(* CODESYS project Parcial2_CPI.project

Project tree, tasks and I/O mapping:
  Device : CODESYS Control Win V3 x64, 3S - Smart Software Solutions GmbH, version 3.5.17.10
    application Application
      libraries: Standard, * (System); CmpBitmapPool, * (System); Util, * (System)
      task MainTask (cyclic, interval t#20ms, priority 1) calls PLC_PRG
      task Simu (cyclic, interval t#20ms, priority 1) calls POU, BOTTLE_SIM
      task VISU_TASK (cyclic, interval 100 ms, priority 31) calls VisuElems.Visu_Prg
      global variables GVL
      program PLC_PRG [ST]
      SIMULACION/
        program BOTTLE_SIM [ST]
        image pool ImagePool
        OBJECTS_METHODS/
          data type BOTTLE_structure
          function colision_detection [ST]
          function modulo [ST]
        program POU [ST]
      visualisation Visualization
      Symbols
      function block AUTO_BF [ST]
      function block MANUAL_BF [ST]
    Ethernet : Ethernet, 3S - Smart Software Solutions GmbH, version 3.5.17.0
        settings: IPAddress = [10,70,28,96]; SubnetMask = [255,255,224,0]; GatewayAddress = [10,70,0,1]; MACAddress = [16#F8,16#5E,16#A0,16#06,16#18,16#05]; NetworkInterfaceName = 'Wi-Fi'; NetworkInterfaceName = "Wi-Fi"; SaveCommunicationSettings = FALSE
      ModbusTCP_Slave_Device : ModbusTCP Slave Device, 3S - Smart Software Solutions GmbH, version 3.5.17.0
          input  Application.PLC_PRG.BOTON_STOP : BOOL  // Registros Holding.Registros Holding.Bit0
          input  Application.PLC_PRG.BOTON_MANUAL : BOOL  // Registros Holding.Registros Holding.Bit1
          input  Application.PLC_PRG.BOTON_AUTO : BOOL  // Registros Holding.Registros Holding.Bit2
          input  Application.BAC1_HMI : BOOL  // Registros Holding.Registros Holding.Bit3
          input  Application.BAC2_HMI : BOOL  // Registros Holding.Registros Holding.Bit4
          input  Application.BABanda_HMI : BOOL  // Registros Holding.Registros Holding.Bit5
          input  Application.BAProducto_HMI : BOOL  // Registros Holding.Registros Holding.Bit6
          input  Application.BAMezclador_HMI : BOOL  // Registros Holding.Registros Holding.Bit7
          input  Application.BADosificacion_HMI : BOOL  // Registros Holding.Registros Holding.Bit8
          input  Application.BOTTLE_SIM.agregar : BOOL  // Registros Holding.Registros Holding.Bit9
          input  Application.BOTTLE_SIM.eliminar : BOOL  // Registros Holding.Registros Holding.Bit10
          output Application.PLC_PRG.PARADA : BOOL  // Registros Input.Registros Input.Bit0
          output Application.PLC_PRG.MANUAL : BOOL  // Registros Input.Registros Input.Bit1
          output Application.PLC_PRG.AUTO : BOOL  // Registros Input.Registros Input.Bit2
          output Application.BAC1_HMI : BOOL  // Registros Input.Registros Input.Bit3
          output Application.BAC2_HMI : BOOL  // Registros Input.Registros Input.Bit4
          output Application.BABanda_HMI : BOOL  // Registros Input.Registros Input.Bit5
          output Application.BAProducto_HMI : BOOL  // Registros Input.Registros Input.Bit6
          output Application.BAMezclador_HMI : BOOL  // Registros Input.Registros Input.Bit7
          output Application.BADosificacion_HMI : BOOL  // Registros Input.Registros Input.Bit8
          unmapped channels: Registros Holding, Registros Input
  libraries: VisuSymbols, 3.5.17.0 (System)
  text list GlobalTextList
  5ce3da45-db07-42e7-a21c-a00fff4ed8f6|imagenes\P1.png
  5ce3da45-db07-42e7-a21c-a00fff4ed8f6|imagenes\P2.png
  5ce3da45-db07-42e7-a21c-a00fff4ed8f6|imagenes\P3.png
  5ce3da45-db07-42e7-a21c-a00fff4ed8f6|imagenes\P4.png
  5ce3da45-db07-42e7-a21c-a00fff4ed8f6|imagenes\P5.png
  5ce3da45-db07-42e7-a21c-a00fff4ed8f6|imagenes\P6.png
  5ce3da45-db07-42e7-a21c-a00fff4ed8f6|imagenes\WaterEmpty.png
  5ce3da45-db07-42e7-a21c-a00fff4ed8f6|imagenes\WaterFilled.png
  5ce3da45-db07-42e7-a21c-a00fff4ed8f6|imagenes\banda.png
  5ce3da45-db07-42e7-a21c-a00fff4ed8f6|imagenes\Cilindro.png
  5ce3da45-db07-42e7-a21c-a00fff4ed8f6|imagenes\Fence.png
  5ce3da45-db07-42e7-a21c-a00fff4ed8f6|imagenes\fondo.png
  5ce3da45-db07-42e7-a21c-a00fff4ed8f6|imagenes\prod2.png
  5ce3da45-db07-42e7-a21c-a00fff4ed8f6|imagenes\prod3.png
  5ce3da45-db07-42e7-a21c-a00fff4ed8f6|imagenes\prod1.png
*)

// Device/Application/SIMULACION/OBJECTS_METHODS/BOTTLE_structure
TYPE BOTTLE_structure :
STRUCT
	empty : BOOL := TRUE; // solid image box
	filled : BOOL := TRUE; // glued image box
	
	pos_x: INT := 0; // x position
	posr_x: REAL := 0; // x position
	
	mvx: REAL := 0.3; // velocidad de movimiento en x
	vx: REAL; // velocidad en x
	
	t_llenado: TON;
END_STRUCT
END_TYPE

// Device/Application/GVL
VAR_GLOBAL
	//MOTORES TRIFASICOS
	BAProducto: BOOL := FALSE; // Señal para encender el motoreductor trifasico elevador del producto
	BAMezclador: BOOL := FALSE; // Señal para encender el motoreductor trifasico de mezclado en la tolva
	BADosificacion: BOOL := FALSE; // Señal para encender el motoreductor trifasico de giro del tornillo de dosificación
	BABanda: BOOL := FALSE; // Señal para encender el motoreductor trifasico de la banda transportadora
	
	//CILINDRO 1 (QUE DETIENE LOS RECIPIENTES QUE VAN A ENTRAR AL PUNTO DE DOSIFICACIÓN)
	BAC1 : BOOL := FALSE; // Señal de avance para el cilindro 1
	SFC1 : BOOL; // Señal de posición final para el cilindro 1
	SIC1 : BOOL; // Señal de posición inicial para el cilindro 1
	
	//CILINDRO 2 (QUE DETIENE EL RECIPIENTE EN EL PUNTO DE DOSIFICACIÓN)
	BAC2 : BOOL := FALSE; // Señal de avance para el cilindro 2
	SFC2 : BOOL; // Señal de posición final para el cilindro 2
	SIC2 : BOOL; // Señal de posición inicial para el cilindro 2
	
	//SENSOR DE PRESENCIA
	SL: BOOL := FALSE; //Sensor de botella en la zona de llenado
	
	//SENSOR DE NIVEL
	NT: INT; //Sensor de 10 bits del nivel de la tolva 
	NTD: BOOL; //Sensor digital del nivel de la tolva (activo cuando el nivel es mayor a 95%)
	
	//HMI
	BAC1_HMI: BOOL;
	BAC2_HMI: BOOL;
	BAProducto_HMI: BOOL;
	BAMezclador_HMI: BOOL;
	BADosificacion_HMI: BOOL;
	BABanda_HMI: BOOL;
	
END_VAR

// Device/Application/PLC_PRG
PROGRAM PLC_PRG
VAR

	PARADA: BOOL := TRUE;
	MANUAL: BOOL;
	AUTO: BOOL;
	BOTON_STOP: BOOL;
	BOTON_MANUAL: BOOL;
	BOTON_AUTO: BOOL;
	
	AUTO1 : AUTO_BF;
	MANUAL1 : MANUAL_BF;
	
END_VAR


IF PARADA AND BOTON_MANUAL THEN
	PARADA := FALSE;
	AUTO := FALSE;
	MANUAL:= TRUE;
	
ELSIF MANUAL AND BOTON_AUTO THEN
	PARADA := FALSE;
	MANUAL:= FALSE;
	AUTO := TRUE;

ELSIF MANUAL AND BOTON_STOP THEN
	PARADA := TRUE;
	AUTO := FALSE;
	MANUAL:= FALSE;

ELSIF AUTO AND BOTON_STOP THEN
	PARADA := TRUE;
	AUTO := FALSE;
	MANUAL:= FALSE;
	
ELSIF PARADA AND BOTON_AUTO THEN
	PARADA := FALSE;
	AUTO := TRUE;
	MANUAL:= FALSE;
	
END_IF

IF PARADA THEN
	BAProducto := FALSE;
	BAMezclador := FALSE;
	BADosificacion := FALSE;
	BABanda := FALSE;
	BAC1 := FALSE;
	BAC2 := FALSE;
	SL := FALSE;
	
ELSIF MANUAL THEN
	MANUAL1();

ELSIF AUTO THEN
	AUTO1();
	
END_IF

END_PROGRAM

// Device/Application/AUTO_BF
FUNCTION_BLOCK AUTO_BF
VAR_INPUT
END_VAR
VAR_OUTPUT
END_VAR
VAR
	
	ON: BOOL := FALSE; //Encender sistema
	STOP: BOOL := FALSE; //Detener botella
	FILL_BOTTLE: BOOL := FALSE; //Llenar botella
	TAKEOUT_BOTTLE: BOOL := FALSE; //Sacar botella de palancas
	FILL_HOPPER: BOOL := FALSE; //Llenar tolva
	NEXT: BOOL := FALSE; //Dejar pasar botella para llenar
	
	TIMER: TON;
	TIMER_RUN_TIME: TIME := T#3S;
	TIMER_RUN: BOOL :=FALSE;
	
	TIMER2 : TON;
	TIMER_RUN_TIME2: TIME := T#1S;
	TIMER_RUN2: BOOL :=FALSE;
	
END_VAR


TIMER(IN:=TIMER_RUN,PT:=TIMER_RUN_TIME);

TIMER2(IN:=TIMER_RUN2,PT:=TIMER_RUN_TIME2);

IF BABanda = FALSE THEN
	ON := TRUE;
END_IF

// PRIMER ESTADO
IF ON = TRUE THEN
	BABanda := TRUE;
	BAMezclador := TRUE;
	BAC2 := TRUE;
	ON := FALSE;
	NEXT := TRUE;
END_IF

// SEGUNDO ESTADO
IF NEXT = TRUE THEN
	BAC2 := TRUE;
	BAC1 := FALSE;
	BAProducto := FALSE;
	IF SL = TRUE THEN
		NEXT := FALSE;
		STOP := TRUE;
	END_IF
END_IF

// TERCER ESTADO
IF STOP = TRUE THEN
	BAC1 := TRUE;
	IF BAC1 = TRUE AND BAC2 = TRUE THEN
		STOP := FALSE;
		FILL_BOTTLE := TRUE;
	END_IF
END_IF

// CUARTO ESTADO
IF FILL_BOTTLE = TRUE THEN
	IF NT = 1023 AND SL = TRUE THEN
		BADosificacion := TRUE;
	ELSIF NT = 972 AND SL = TRUE THEN
		BADosificacion := FALSE;
		FILL_BOTTLE := FALSE;
		TAKEOUT_BOTTLE := TRUE;
	END_IF
END_IF

// QUINTO ESTADO
IF TAKEOUT_BOTTLE = TRUE THEN
	TIMER_RUN := TRUE;
	BAC2 := FALSE;
	IF TIMER.Q = TRUE THEN
		TIMER_RUN := FALSE;
		TAKEOUT_BOTTLE := FALSE;
	END_IF
	FILL_HOPPER := TRUE;
END_IF

// SEXTO ESTADO
IF FILL_HOPPER = TRUE THEN
	TIMER_RUN2 := TRUE;
	BAProducto := TRUE;
	IF TIMER2.Q = TRUE THEN
		TIMER_RUN2 := FALSE;
		BAProducto := FALSE;
		FILL_HOPPER := FALSE;
		NEXT := TRUE;
	END_IF
END_IF

END_FUNCTION_BLOCK

// Device/Application/MANUAL_BF
FUNCTION_BLOCK MANUAL_BF
VAR_INPUT
END_VAR
VAR_OUTPUT
END_VAR
VAR
END_VAR


BAProducto := BAProducto_HMI;
BAMezclador := BAMezclador_HMI;
BADosificacion := BADosificacion_HMI;
BABanda := BABanda_HMI;
BAC1 := BAC1_HMI;
BAC2 := BAC2_HMI;

END_FUNCTION_BLOCK

// Device/Application/SIMULACION/POU
PROGRAM POU
VAR
	Intervalo : INT := 20; //ms, Debe corresponder al intervalo de ejecución de la tarea Simu 	
	
	NTolvaMax : REAL := 100; //Nivel maximo de la tolva
	NTolva : REAL := 100; //Nivel de la tolva
	TTolva : REAL := 5; // Tiempo que le toma a la tolva vaciarse
	VLTolva : REAL := NTolva*(intervalo*1E-3)/TTolva; // Velocidad de llenado de la tolva
	VVTolva : REAL := NTolva*(intervalo*1E-3)/TTolva/10; // Velocidad de vaciado de la tolva
	
	CProducto: WORD := 4; //Valor maximo del contador para la animacion
	AProducto: WORD := 0; //Valor actual del contador
	ANIProducto: CTU; //Contador para generar la animacion
	BLKProducto: BLINK; //señal de conteo
	TProducto: TIME := T#0.3S; //tiempo de transición del blink 
	
	BLKBanda: BLINK;
	TBanda: TIME:= T#0.5S;
	
	
	PYIC1 : INT := 506; // posicion inicial en y del cilindro 1
	PYFC1 : INT := 490; // posicion final en y del cilindro 1
	PYC1 : INT; //posicion en y del cilindro 1
	TCI1: TON; //timer para retardar la señal de posición inicial del cilindro 1
	TCF1: TON; //timer para retardar la señal de posición final del cilindro 1
	TIMERC1: TIME:= T#0.3S; //tiempo de retardo para activar las señales de los sensores de posición del cilindro 1
	
	PYIC2 : INT := 506; // posicion inicial en y del cilindro 1
	PYFC2 : INT := 490; // posicion final en y del cilindro 1
	PYC2 : INT; //posicion en y del cilindro 1
	TCI2: TON; //timer para retardar la señal de posición inicial del cilindro 2
	TCF2: TON; //timer para retardar la señal de posición final del cilindro 2
	TIMERC2: TIME:= T#0.3S; //tiempo de retardo para activar las señales de los sensores de posición del cilindro 2
END_VAR

//TOLVA
//Llenado y vaciado de la tolva
IF BAProducto AND NTolva < NTolvaMax THEN
	NTolva := MIN(NTolva + VLTolva, NTolvaMax);
END_IF
BLKProducto(ENABLE:=BADosificacion, TIMELOW:=TProducto, TIMEHIGH:=TProducto);
ANIProducto(CU:=BLKProducto.OUT,RESET:=ANIProducto.Q OR NOT(BADosificacion) OR NTolva = 0,PV := CProducto); 
IF BADosificacion THEN 
	 IF NTolva > 0 THEN
		NTolva := MAX(NTolva - VVTolva, 0);
	END_IF
END_IF
NT:= TO_INT(NTolva/NTolvaMax*1023);
NTD := NTolva/NTolvaMax > 0.95;


//cilindro 1
//Movimiento del cilindro 1
TCF1(IN:=BAC1,PT:=TIMERC1);
TCI1(IN:=NOT BAC1,PT:=TIMERC1);
IF BAC1 THEN
	PYC1 := PYFC1-PYIC1;
	IF TCF1.Q THEN
		//Señales del cilindro 1
		SFC1 := TRUE;
		SIC1 := FALSE;
	END_IF
ELSE
	PYC1 := 0;
	IF TCI1.Q THEN
		//Señales del cilindro 1
		SFC1 := FALSE;
		SIC1 := TRUE;
	END_IF
END_IF

//cilindro 2
//Movimiento del cilindro 2
TCF2(IN:=BAC2,PT:=TIMERC2);
TCI2(IN:=NOT BAC2,PT:=TIMERC2);
IF BAC2 THEN
	PYC2 := PYFC2-PYIC2;
	IF TCF2.Q THEN
		//Señales del cilindro 2
		SFC2 := TRUE;
		SIC2 := FALSE;
	END_IF
ELSE
	PYC2 := 0;
	IF TCI2.Q THEN
		//Señales del cilindro 2
		SFC2 := FALSE;
		SIC2 := TRUE;
	END_IF
END_IF


//BANDA
BLKBanda(ENABLE:=BABanda, TIMELOW:=TBanda, TIMEHIGH:=TBanda);

END_PROGRAM

// Device/Application/SIMULACION/BOTTLE_SIM
PROGRAM BOTTLE_SIM
VAR
	
	agregar: BOOL; //variable que indica que se debe agregar una botella
	agregar_ant: BOOL := FALSE; //variable para detectar el cambio de estado en el boton agregar
	eliminar: BOOL; //variable que indica que se debe eliminar una botella
	eliminar_ant: BOOL := FALSE; //variable para detectar el cambio de estado en el boton eliminar
	bottles : ARRAY[0..4] OF BOTTLE_structure;
	
	SL_any: BOOL; //variable auxiliar para indicar que alguna botella esta en la zona de llenado
	
	total_bottles: INT := 5; //Botellas totales
	bot_agregadas: INT := 0; //Botellas agregadas
	
	b_add : BOOL;
	i : INT;
	k : INT;
	i_add : INT := 0; //indice de la siguiente botella a agregar
	i_delete : INT := 0; //indice de la siguiente botella a eliminar
	
	ancho_botella : INT := 19;
	sep_botellas : INT := 20; //separación entre botellas a la hora de agregar más
	
	//Posiciones y dimensiones
	bot_init_x : INT := 262; //posicion x inicial de las botella
	bot_init_y : INT := 478; //posicion y inicial de las botella
	bot_x: REAL; //posicion x de la botella en la visualización
	
	cil1_x: INT := 467; //posicion x del cilindro 1
	cil2_x: INT := 497; //posicion x del cilindro 2
	cil_ancho: INT := 6; //ancho de un cilindro
	
	llenado_init: INT := 469; //posicion x de inicio de la zona de llenado
	llenado_fin: INT := 485; //posicion x de fin de la zona de llenado
	
	banda_fin: INT := 950; //posicion donde la banda termina
END_VAR



IF agregar AND NOT agregar_ant AND bot_agregadas < total_bottles THEN
	b_add := TRUE;
	IF bot_agregadas > 0 THEN
		k := modulo(i_add-1,total_bottles);
		b_add := bottles[k].pos_x > ancho_botella + sep_botellas;
	END_IF
	IF b_add then
		bottles[i_add].pos_x := 0;
		bottles[i_add].posr_x := 0;
		bottles[i_add].empty := FALSE;
		bottles[i_add].filled := TRUE;
		bot_agregadas := bot_agregadas + 1;
		i_add := (i_add+1) MOD total_bottles;
		k:=1;
	END_IF
END_IF
agregar_ant := agregar;

IF eliminar AND NOT eliminar_ant AND bot_agregadas > 0 THEN
	bottles[i_delete].empty := TRUE;
	bottles[i_delete].filled := TRUE;
	bot_agregadas := bot_agregadas - 1;
	i_delete := (i_delete+1) MOD total_bottles;
END_IF
eliminar_ant := eliminar;

SL_any := FALSE;
FOR i := 0 to total_bottles-1 do
	IF NOT bottles[i].empty OR NOT bottles[i].filled THEN
		bot_x := bottles[i].posr_x+bot_init_x;
		bottles[i].vx := 0;
		
		//Desplazamiento cuando la banda esta encendida
		IF BABanda THEN
			bottles[i].vx := bottles[i].mvx;
		END_IF
		
		//colision con cilindro 1
		IF colision_detection(bot_x, ancho_botella, bottles[i].mvx,cil1_x) AND SFC1 THEN
			bottles[i].vx := 0;
		END_IF
		
		//colision con cilindro 2
		IF colision_detection(bot_x, ancho_botella, bottles[i].mvx,cil2_x) AND SFC2 THEN
			bottles[i].vx := 0;
		END_IF
		
		//colision con botella anterior
		IF colision_detection(bottles[i].pos_x, ancho_botella, bottles[i].mvx, bottles[modulo(i-1, total_bottles)].pos_x-sep_botellas) AND
				(NOT bottles[modulo(i-1, total_bottles)].empty OR NOT bottles[modulo(i-1, total_bottles)].filled)THEN
			bottles[i].vx := 0;
		END_IF
		
		//botella en zona de llenado
		if bot_x >= llenado_init and bot_x <= llenado_fin then
			SL_any := TRUE;
			bottles[i].t_llenado(IN:=BADosificacion, PT:=T#2s);	
		END_IF
		
		//tiempo de dosificación alcanzado
		IF bottles[i].t_llenado.Q then
			bottles[i].empty := TRUE;
			bottles[i].filled := FALSE;
			bottles[i].t_llenado(IN:=FALSE, PT:=T#4S);
		END_IF
		
		//salida de la botella
		IF bot_x >= banda_fin THEN
			bottles[i].empty := TRUE;
			bottles[i].filled := TRUE;
			bot_agregadas := bot_agregadas - 1;
			i_delete := (i_delete+1) MOD total_bottles;
		END_IF
		
		bottles[i].posr_x := bottles[i].posr_x + bottles[i].vx;
		
		
	END_IF
	
	bottles[i].pos_x := TRUNC_INT(bottles[i].posr_x);
END_FOR

SL := SL_any;

END_PROGRAM

// Device/Application/SIMULACION/OBJECTS_METHODS/modulo
FUNCTION modulo : INT
VAR_INPUT
	x: INT;
	y: INT;
END_VAR
VAR
END_VAR

IF x>=0 THEN
	modulo := x MOD y;
ELSE
	modulo := TO_INT( (y*(ABS(FLOOR(x/y))+1)+x) MOD y);
END_IF

END_FUNCTION

// Device/Application/SIMULACION/OBJECTS_METHODS/colision_detection
FUNCTION colision_detection : BOOL
VAR_INPUT
	pos: REAL; //Posicion del objeto 
	ancho: REAL; //anchura del objeto
	vel: REAL; //Velocidad del objeto
	pos_obst_init: REAL; //posicion donde comienza el obstaculo
END_VAR
VAR
END_VAR

colision_detection := pos + vel < pos_obst_init AND pos +ancho+ vel > pos_obst_init;

END_FUNCTION

// Device/Application/Visualization
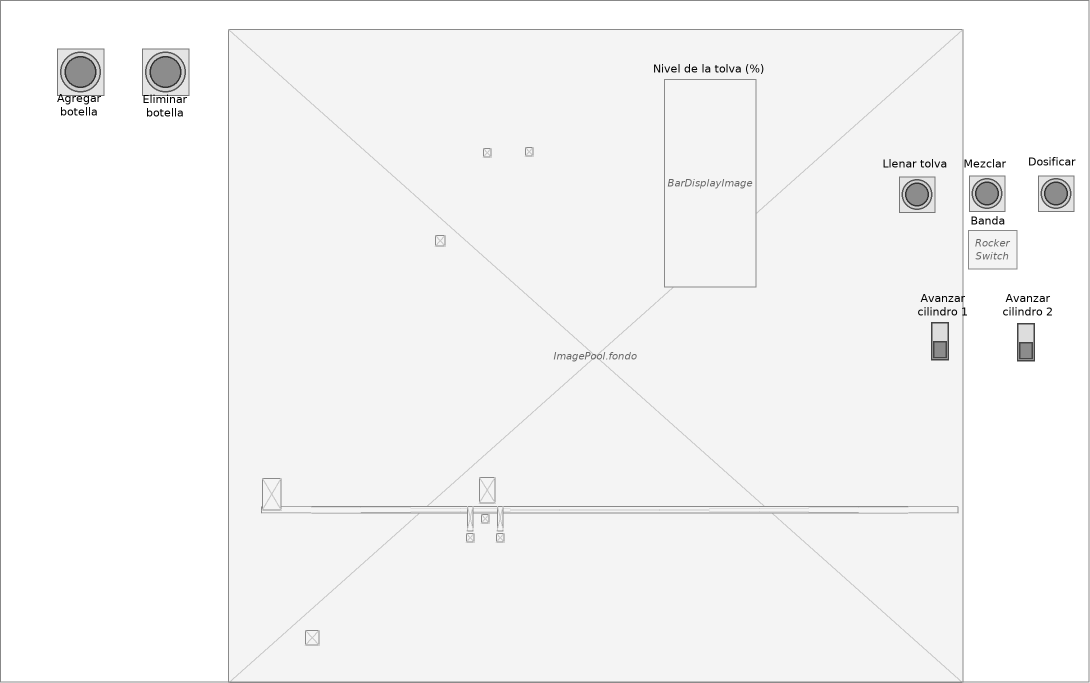
VISUALIZATION Visualization  // 1090x683
    PushSwitchLed (57,46 47x52), variable: BOTTLE_SIM.agregar, behaviour: TAP, style: Switch-PushSwitchLed-Gray
    Label (41,84 76x42), "Agregar botella"
    PushSwitchLed (142,46 47x52), variable: BOTTLE_SIM.eliminar, behaviour: TAP, style: Switch-PushSwitchLed-Gray
    Label (127,87 76x38), "Eliminar botella"
    Image (228,29 735x654), image: ImagePool.fondo
    Image (261,506 697x7), invisible if: POU.BLKBanda.OUT, image: ImagePool.banda
    BarDisplayImage (664,79 92x208), value: POU.NTolva, style: BarDisplayImage-Gray, scale format: %.0f, scale 0..100
    Label (634,54 150x30), "Nivel de la tolva (%)"
    PushSwitch (1038,171 36x45), variable: BADosificacion, behaviour: TOGGLE, style: Switch-PushSwitch-Gray
    Image (305,630 14x15), invisible if: NOT BAProducto, image: ImagePool.boton_verde
    Image (483,148 8x9), invisible if: NOT BADosificacion, image: ImagePool.boton_verde
    Image (525,147 8x9), invisible if: NOT BAMezclador, image: ImagePool.boton_verde
    Image (466,533 8x9), invisible if: SIC1, image: ImagePool.boton_verde
    Image (496,533 8x9), invisible if: SIC2, image: ImagePool.boton_verde
    Image (481,514 8x9), invisible if: not SL, image: ImagePool.boton_verde
    Label (1014,147 76x30), "Dosificar"
    PushSwitch (899,172 36x45), variable: BAProducto, behaviour: TOGGLE, style: Switch-PushSwitch-Gray
    Label (871,149 88x30), "Llenar tolva"
    PushSwitch (969,171 36x45), variable: BAMezclador, behaviour: TAP, style: Switch-PushSwitch-Gray
    Label (947,149 76x30), "Mezclar"
    RockerSwitch (968,230 49x39), variable: BABanda, behaviour: TOGGLE, style: Switch-RockerSwitch-Gray
    Label (950,206 76x30), "Banda"
    Image (481,477 10x14), invisible if: NOT(POU.ANIProducto.CV=1), image: ImagePool.prod1
    Image (481,479 10x16), invisible if: NOT(POU.ANIProducto.CV=2), image: ImagePool.prod2
    Image (479,477 16x26), invisible if: NOT(POU.ANIProducto.CV=3), image: ImagePool.prod3
    Image (262,478 19x32), invisible if: BOTTLE_SIM.bottles[0].empty, image: ImagePool.WaterEmpty
        p3560616238: BOTTLE_SIM.bottles[0].pos_x
    Image (467,506 6x25), image: ImagePool.Cilindro
        p2738717112: POU.PYC1
    Image (497,506 6x25), image: ImagePool.Cilindro
        p2738717112: POU.PYC2
    Label (899,278 88x54), "Avanzar cilindro 1"
    Label (984,278 88x54), "Avanzar cilindro 2"
    Image (262,478 19x32), invisible if: BOTTLE_SIM.bottles[0].filled, image: ImagePool.WaterFilled
        p3560616238: BOTTLE_SIM.bottles[0].pos_x
    Image (262,478 19x32), invisible if: BOTTLE_SIM.bottles[1].empty, image: ImagePool.WaterEmpty
        p3560616238: BOTTLE_SIM.bottles[1].pos_x
    Image (262,478 19x32), invisible if: BOTTLE_SIM.bottles[1].filled, image: ImagePool.WaterFilled
        p3560616238: BOTTLE_SIM.bottles[1].pos_x
    Image (262,478 19x32), invisible if: BOTTLE_SIM.bottles[3].empty, image: ImagePool.WaterEmpty
        p3560616238: BOTTLE_SIM.bottles[3].pos_x
    Image (262,478 19x32), invisible if: BOTTLE_SIM.bottles[3].filled, image: ImagePool.WaterFilled
        p3560616238: BOTTLE_SIM.bottles[3].pos_x
    Image (262,478 19x32), invisible if: BOTTLE_SIM.bottles[2].empty, image: ImagePool.WaterEmpty
        p3560616238: BOTTLE_SIM.bottles[2].pos_x
    Image (262,478 19x32), invisible if: BOTTLE_SIM.bottles[2].filled, image: ImagePool.WaterFilled
        p3560616238: BOTTLE_SIM.bottles[2].pos_x
    Image (262,478 19x32), invisible if: BOTTLE_SIM.bottles[4].empty, image: ImagePool.WaterEmpty
        p3560616238: BOTTLE_SIM.bottles[4].pos_x
    Image (262,478 19x32), invisible if: BOTTLE_SIM.bottles[4].filled, image: ImagePool.WaterFilled
        p3560616238: BOTTLE_SIM.bottles[4].pos_x
    Image (435,235 10x11), invisible if: NOT NTD, image: ImagePool.boton_verde
    DipSwitch (921,322 38x38), variable: BAC1, behaviour: TOGGLE, style: Switch-DipSwitch-Gray
    DipSwitch (1007,323 38x38), variable: BAC2, behaviour: TOGGLE, style: Switch-DipSwitch-Gray
END_VISUALIZATION
